FUNCTION_BLOCK FB_JoystickInputScaling_1
// LREAL: Long Real decimal number
// INT: [-32768, 32767]	
// BOOL: True/False

// Input variables (value set in PRG)
VAR_INPUT
	bEnable 				: BOOL;
	nRawInput 				: INT;
	fMaxValue 				: LREAL;
	fMaxInputValue			: LREAL;
	fMinInputValue 			: LREAL;
	fNeutralInputValue  	: LREAL;
	fNeutralDeadband		: LREAL;
END_VAR

// Output variables
VAR_OUTPUT
	fOutput : LREAL;
END_VAR

// Variables
VAR			
	fRawInput : LREAL;		// Raw input value
	fTempInput : LREAL; 	// Temporary input
	fTempOutput : LREAL; 	// Temporary output

	fMaxOutputValue  		: LREAL := 1.0;
	fMinOutputValue  		: LREAL := -1.0;
	fNeutralOutputValue  	: LREAL := 0.0;
END_VAR

// Crane is only supported for movement in the y-axis (up/down)

fRawInput := INT_TO_LREAL(nRawInput); 			// Converts input to decimal number
fTempInput := fRawInput - fNeutralInputValue; 	// Defines neutral point 

IF fTempInput > fNeutralDeadband THEN 									// If input is above the neutral deadband (positive y) 
	fTempOutput := fTempInput/(fMaxInputValue - fNeutralInputValue); 	// Scales positive movement [0,1]
ELSIF fTempInput < -fNeutralDeadband THEN 								// If input is below the neutral deadband (negative y)
	fTempOutput := fTempInput/(fNeutralInputValue - fMinInputValue); 	// Scales negative movement [-1,0]
ELSE
	fTempOutput := 0.0; 			// If joystick is inside deadzone, fTempOutput = 0
END_IF

IF NOT(bEnable) THEN 				// If bEnable is not true, set fOutput = 0
	fOutput := 0.0;
ELSE
	fOutput := LIMIT(fMinOutputValue * fMaxValue, fTempOutput * fMaxValue, fMaxOutputValue* fMaxValue); 
	// Calculates output signal within safety limits (Min, Output, Max)
END_IF

END_FUNCTION_BLOCK

(* stored: Version 1.1.0.1
   POU FB_JoystickInputScaling_1: Id {567a891a-c9cb-4c8d-af8e-f47a632b067b}, SpecialFunc None *)
